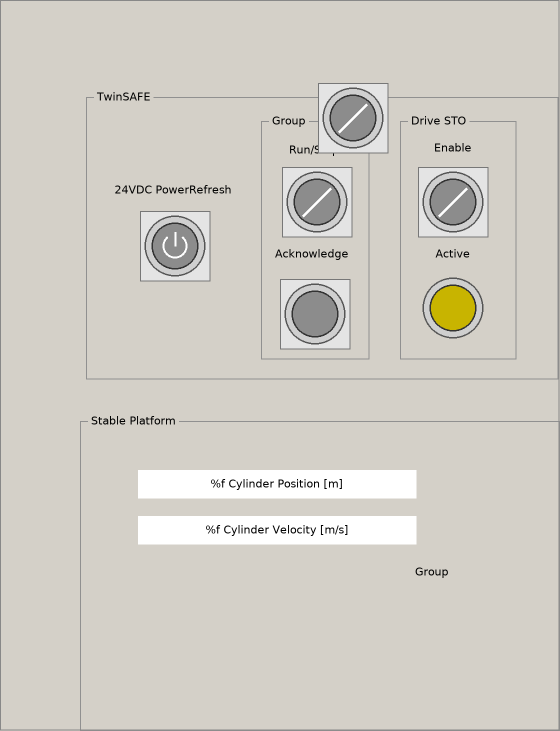
VISUALIZATION HMI  // 560x731
    GroupBox (86,89 472x290), "TwinSAFE"
        PowerSwitch (54,122 70x70), variable: GVL_Safety_AXIS4.bWinchMotor24vDisable, behaviour: TAP, style: Switch-PowerSwitch-Gray
        Label (12,86 150x30), "24VDC PowerRefresh"
        Label (268,468 156x30), "Group"
        Label (150,46 156x30), "Run/Stop"
        Label (148,150 156x30), "Acknowledge"
        GroupBox (175,24 108x246), "Group"
            RotarySwitch (21,54 70x70), variable: GVL_Safety_AXIS4.TwinSafeGroupRunStop, behaviour: TOGGLE, style: Switch-RotarySwitch-Gray
            PushSwitch (19,166 70x70), variable: GVL_Safety_AXIS4.TwinSafeGroupComErrAck, behaviour: TAP, style: Switch-PushSwitch-Gray
        Lamp1 (170,918 70x70), variable: GVL_Safety_AXIS4.ChA_STO_Active, style: Lamp-Lamp1-Yellow
        GroupBox (314,24 116x246), "Drive STO"
            RotarySwitch (-82,-30 70x70), behaviour: TOGGLE, style: Switch-RotarySwitch-Gray
            RotarySwitch (18,54 70x70), variable: GVL_Safety_AXIS4.ChA_STO_Enable, behaviour: TOGGLE, style: Switch-RotarySwitch-Gray
            Lamp1 (18,160 70x70), variable: GVL_Safety_AXIS4.ChA_STO_Active, style: Lamp-Lamp1-Yellow
        Label (292,44 150x30), "Enable"
        Label (292,150 150x30), "Active"
    GroupBox (80,413 480x318), "Stable Platform"
        Textfield (57,56 280x30), "%f Cylinder Position [m]", text variable: G_StablePlatformScaledIO.fPistonPosition
        Textfield (57,102 280x30), "%f Cylinder Velocity [m/s]", text variable: G_StablePlatformScaledIO.fPistonVelocity
END_VISUALIZATION

(* stored: Version 1.1.0.1, ProductVersion 3.1.4024.12
   Visu HMI: Id {4fc9a593-5585-4c7b-9c87-b23c76f2039c} *)
